// TIA Portal project "DawidKania_OptimizeLReal" (V14)

(* hardware
DEVICE "S7-1200 station_1"  S7-1200 Station
   slot 0: "Rack_0"  S7-1200 Rack  Rack  V1.0
   slot 1: "PLC_1"  CPU 1214C DC/DC/DC  6ES7 214-1AG31-0XB0  V3.0
*)

// ===== PLC "PLC_1"  CPU 1214C DC/DC/DC =====

FUNCTION "OptimizedFunction" : LReal   // FC1, SCL
{ S7_Optimized_Access := 'TRUE' }
VERSION : 0.1
   VAR_INPUT
      x1 : LReal;
      x2 : LReal;
   END_VAR
BEGIN
   // find minimum of function
   // y = x1 ^2 - 6 *x1 ^2.*x2 - 20 *x1 + 3 *x2 ^2 + 3 *x1 ^4 + 109


   #OptimizedFunction := #x1 ** LREAL#2.0 - LREAL#6.0 * #x1 ** LREAL#2.0 * #x2
   - LREAL#20.0 * #x1 + LREAL#3.0 * #x2 ** LREAL#2.0
   + LREAL#3.0 * #x1 ** LREAL#4.0 + lREAL#109.0;
END_FUNCTION

FUNCTION "GradientSearchMin" : LReal   // FC2, SCL
{ S7_Optimized_Access := 'TRUE' }
VERSION : 0.1
   VAR_INPUT
      x01 : LReal;
      x02 : LReal;
      iter : Int;
   END_VAR
   VAR_TEMP
      x1 : LReal;
      x2 : LReal;
      delta : LReal;
      alpha : LReal;
      y : LReal;
      y1 : LReal;
      y2 : LReal;
      dy_dx1 : LReal;
      dy_dx2 : LReal;
   END_VAR
BEGIN

   #delta := LREAL#0.001;
   #alpha := LREAL#1.0;

   #x1 := #x01;
   #x2 := #x02;

   WHILE #iter >= 0 DO
       #iter := #iter - 1;

       // calculate gradient
       #y := "OptimizedFunction"(x1:=#x1, x2:=#x2);
       #y1 := "OptimizedFunction"(x1:=#x1 + #delta, x2:=#x2);
       #y2 := "OptimizedFunction"(x1:=#x1, x2:=#x2 + #delta);

       #dy_dx1 := (#y1 - #y) / #delta;
       #dy_dx2 := (#y2 - #y) / #delta;

       #x1 := #x1 - #alpha * #dy_dx1;
       #x2 := #x2 - #alpha * #dy_dx2;

   END_WHILE;

   #GradientSearchMin := "OptimizedFunction"(x1:=#x1, x2:=#x2);
END_FUNCTION

ORGANIZATION_BLOCK "Main"   // OB1, SCL, ProgramCycle
TITLE = "Main Program Sweep (Cycle)"
{ S7_Optimized_Access := 'TRUE' }
VERSION : 0.1
   VAR_TEMP
      minimum : LReal;
   END_VAR
BEGIN


   #minimum := "GradientSearchMin"(x01:=LREAL#100.0, x02:=LREAL#100.0, iter:=1000);
END_ORGANIZATION_BLOCK